Staubli VAL3: CmdManage.pgx

program CmdManage()
begin
  while true
    //add data received into buffer
    if ststu==true and CmdTotal<20
      CmdBuffer[nWritePt]=datar
      CmdTotal=CmdTotal+1
      nWritePt=nWritePt+1
      if nWritePt>=20
        nWritePt=0
      endIf
      //HERE BELOW IS HIGH PRIORITY OF HOMING ROBOT
      datar=""
      ststu=false
    endIf
    delay(0)
  endWhile
end
